# EPICS autosave request: iocBoot/generic_motors_ioc/dbSave/BP_Hd2_.req
%
% BURT Request File
%
% $(P)BP:Kb:  BPM @ KB mirrors position
%
file assy.req ASSY=$(P)BP:Hd2
file mtr1.req MTR1=$(P)BP:mh2z
file drv1.req DRV1=$(P)BP:H2Z
